{attribute 'GeneratedUsingTerminal: EL4031-0000-0016'}
{attribute addProperty BoxType "EL4031-0000-0016"}
{attribute addProperty Description "EL4031 1Ch. Ana. Output +/-10V, 12bit"}
{attribute addProperty Physics "KK"}
{attribute addProperty Id "AO_OutputsAT %Q*AO_Output_Channel_BA7EBB7C2WcStateAT %I*WcState_0B2B16F91InfoDataAT %I*InfoData_32EB74EA10"}
{attribute addProperty CRC "3024842059"}
{attribute addProperty Size "13"}
TYPE EL4031_B44B6D4B EXTENDS EtcSlaveTerminalBase_947E5A46 :
STRUCT
	{attribute addProperty Name "AO_Outputs"}
	AO_Outputs : AO_Output_Channel_BA7EBB7C;
	{attribute addProperty Name "WcState"}
	WcState : WcState_0B2B16F9;
	{attribute addProperty Name "InfoData"}
	InfoData : InfoData_32EB74EA;
END_STRUCT
END_TYPE

(* stored: Version 1.2.0.0, ProductVersion 3.1.4024.11
   DUT EL4031_B44B6D4B: Id {dee81a1f-43d6-4918-b536-4fa73e2a6f58} *)
